(* PLC project cp_trich, Dassault Systèmes ControlBuild 2024x *)
(* stored: creationDateTime 2023-10-03T11:13:59-01:00 *)

PROGRAM tri_chain.cp_trich
  VAR_INPUT
    ON : BOOL := false;
    run1 : BOOL := false;
    startSensor1 : BOOL := false;
    endSensor1 : BOOL := false;
    run2 : BOOL := false;
    startSensor2 : BOOL := false;
    endSensor2 : BOOL := false;
    run3 : BOOL := false;
    startSensor3 : BOOL := false;
    endSensor3 : BOOL := false;
    sensor1 : BOOL := false;
    sensor2 : BOOL := false;
    sensor3 : BOOL := false;
    endSensor : BOOL := false;
    endSensor4 : BOOL := false;
  END_VAR
  VAR_OUTPUT
    mvt1 : BOOL := false;
    mvt2 : BOOL := false;
    mvt3 : BOOL := false;
    moveToLeft : BOOL := false;
    moveToRight : BOOL := false;
    chainMvt : BOOL := false;
    mvt4 : BOOL := false;
  END_VAR

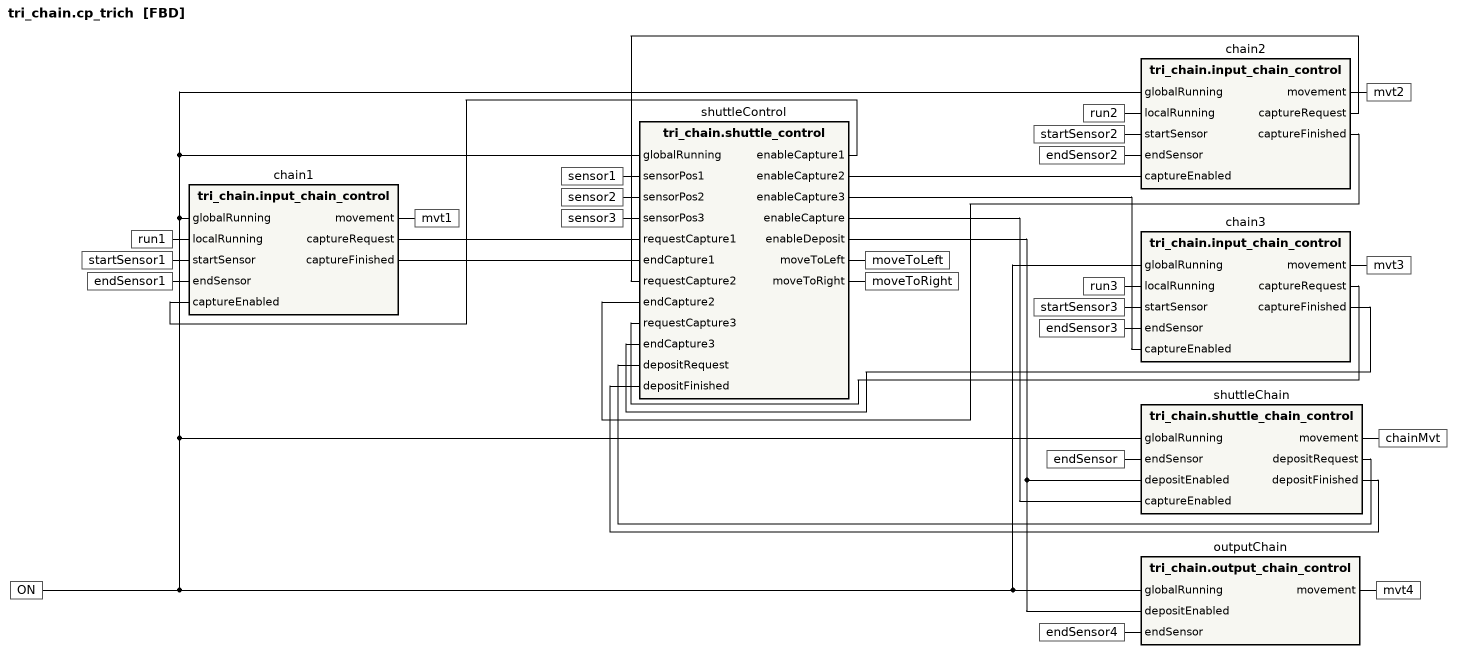
(* FBD diagram, written out as Structured Text *)
chain2(globalRunning := ON, localRunning := run2, startSensor := startSensor2, endSensor := endSensor2, captureEnabled := shuttleControl.enableCapture2);
chain3(globalRunning := ON, localRunning := run3, startSensor := startSensor3, endSensor := endSensor3, captureEnabled := shuttleControl.enableCapture3);
shuttleChain(globalRunning := ON, endSensor := endSensor, depositEnabled := shuttleControl.enableDeposit, captureEnabled := shuttleControl.enableCapture);
shuttleControl(globalRunning := ON, sensorPos1 := sensor1, sensorPos2 := sensor2, sensorPos3 := sensor3, requestCapture1 := chain1.captureRequest, endCapture1 := chain1.captureFinished, requestCapture2 := chain2.captureRequest, endCapture2 := chain2.captureFinished, requestCapture3 := chain3.captureRequest, endCapture3 := chain3.captureFinished, depositRequest := shuttleChain.depositRequest, depositFinished := shuttleChain.depositFinished);
chain1(globalRunning := ON, localRunning := run1, startSensor := startSensor1, endSensor := endSensor1, captureEnabled := shuttleControl.enableCapture1);
mvt1 := chain1.movement;
mvt2 := chain2.movement;
mvt3 := chain3.movement;
moveToLeft := shuttleControl.moveToLeft;
moveToRight := shuttleControl.moveToRight;
chainMvt := shuttleChain.movement;
outputChain(globalRunning := ON, depositEnabled := shuttleControl.enableDeposit, endSensor := endSensor4);
mvt4 := outputChain.movement;
END_PROGRAM
